# B&R Automation Studio project X20AP3x
Automation Studio 4.3.6.57 SP

## Configuration Config1

CPU , AutomationRuntime E3.10, Build 4.1.2, Vc V3.96.2

### Task classes (Cpu.sw)
```
Cyclic#1 (cycle 2000 us, tolerance 0 us):
  CondMon <- ConditionalMonitoring.CondMon.prg
Binaries: ashwd, sysconf, asfw, arconfig, iomap
Libraries: AsFltGen, AsBrStr, runtime, X20AP31x, astime, asieccon
```

### Hardware
```
PLC1 : X20CP1484 v1.1.5.0
  Connector IF2:
    ActivateDevice = 1
    Mode = Manual
    InternetAddress = 10.49.40.222
    SubnetMask = 255.255.255.0
  Connector IF3:
    InaNodeNumber = 1
  Cyclic1Duration = 2000
  Cyclic1Tolerance = 0
  Cyclic2Duration = 10000
  Cyclic2Tolerance = 10000
X20AP3131 : X20AP3131 v1.1.1.0  [SS1 -> X20TB32.SS; SL -> X20BM32.SL1]
  Supervision = off
  EnergyUnit = 1Ws
  ConfigPhaseN = calc
  VoltageWarnLim = 22000
  ZeroCrossing = on
  DisPFmeanT = off
  DisPmeanT = off
  DisQmeanT = off
  DisSmeanT = off
  DisAcEnT = off
  DisReacEnT = off
  DisAppEnT = off
  FlatStreamActivate = on
X20BM32 : X20BM32 v1.0.0.1  [X2X1 -> PLC1.IF6]
X20TB32 : X20TB32 v1.0.0.1
```

### IoMap.iom - PLC1/IoMap.iom
```iecst
(********************************************************************
 * COPYRIGHT -- Bernecker + Rainer
 ********************************************************************
 * Datei: IoMap.iom
 * Autor: hilchenbachc
 * Erstellt: 10. Januar 2014
 ********************************************************************
 * IO-Rangierungsdatei
 ********************************************************************)
VAR_CONFIG
	::CondMon:iomapping.in.InputSequence AT %IB."X20AP3131".InputSequence;
	::CondMon:iomapping.in.RxByte1 AT %IB."X20AP3131".RxByte1;
	::CondMon:iomapping.in.RxByte2 AT %IB."X20AP3131".RxByte2;
	::CondMon:iomapping.in.RxByte3 AT %IB."X20AP3131".RxByte3;
	::CondMon:iomapping.in.RxByte4 AT %IB."X20AP3131".RxByte4;
	::CondMon:iomapping.in.RxByte5 AT %IB."X20AP3131".RxByte5;
	::CondMon:iomapping.in.RxByte6 AT %IB."X20AP3131".RxByte6;
	::CondMon:iomapping.in.RxByte7 AT %IB."X20AP3131".RxByte7;
	::CondMon:iomapping.out.OutputSequence AT %QB."X20AP3131".OutputSequence;
	::CondMon:iomapping.out.EnabEnergy AT %QX."X20AP3131".EnabEnergy;
	::CondMon:iomapping.in.RBTrigDFT AT %IX."X20AP3131".RBTrigDFT;
	::CondMon:iomapping.out.TrigDFT AT %QX."X20AP3131".TrigDFT;
	::condMonData.MainsStatus.WarningPhaseA AT %IX."X20AP3131".WarningPhaseA;
	::condMonData.MainsStatus.WarningPhaseB AT %IX."X20AP3131".WarningPhaseB;
	::condMonData.MainsStatus.WarningPhaseC AT %IX."X20AP3131".WarningPhaseC;
	::condMonData.MainsStatus.LossPhaseA AT %IX."X20AP3131".LossPhaseA;
	::condMonData.MainsStatus.LossPhaseB AT %IX."X20AP3131".LossPhaseB;
	::condMonData.MainsStatus.LossPhaseC AT %IX."X20AP3131".LossPhaseC;
END_VAR
```

## Logical view

Binary libraries used (declarations not repeated): operator, runtime, astime, AsIecCon, AsBrStr, AsFltGen


### Package Logical/ConditionalMonitoring - Energieerfassung

### ConditionalMonitoring.typ - Paket Datentypen
```iecst
TYPE
	CondMonEnergy : 	STRUCT
		SVenergyT : LREAL; (* (Vector Sum) Total Apparent Energy [kWh]*)
	END_STRUCT;
	CondMonPower : 	STRUCT
		SVmeanT : LREAL; (*  (Vector Sum) Total Apparent Power [W]*)
		PmeanT : LREAL; (* Total Active Power [W]*)
		QmeanT : LREAL; (*  Total Reactive Power [W]*)
		PFmeanT : LREAL; (*  Total power factor [1]*)
	END_STRUCT;
	CondMonMainsStatus : 	STRUCT
		frequency : LREAL; (*Netzfrequenz*)
		TresholdWarning : LREAL; (*Spannungsschwelle für Warnung*)
		WarningPhaseA : BOOL;
		WarningPhaseB : BOOL;
		WarningPhaseC : BOOL;
		TresholdLoss : LREAL; (*Spannungsschwelle für Ausfall*)
		LossPhaseA : BOOL;
		LossPhaseB : BOOL;
		LossPhaseC : BOOL;
		MainsOK : BOOL;
	END_STRUCT;
	CondMonRMS : 	STRUCT
		UrmsA : LREAL; (* phase A voltage RMS [V]*)
		UrmsB : LREAL; (* phase B voltage RMS [V]*)
		UrmsC : LREAL; (* phase C voltage RMS [V]*)
		IrmsN : LREAL; (* N Line calculated current RMS [A]*)
		IrmsA : LREAL; (* phase A voltage RMS [A]*)
		IrmsB : LREAL; (* phase B voltage RMS [A]*)
		IrmsC : LREAL; (* phase C voltage RMS [A]*)
	END_STRUCT;
	CondMonData : 	STRUCT
		Rms : CondMonRMS; (*elektrische Effektivwerte*)
		Power : CondMonPower; (*elektrische Leistung*)
		Energy : CondMonEnergy; (*elektrische Arbeit*)
		MainsStatus : CondMonMainsStatus; (*Status des Versorgungsnetzes*)
	END_STRUCT;
END_TYPE
```

### ConditionalMonitoring.var - Paket Variablen
```iecst
VAR
	condMonData : CondMonData; (*Condition Monitoring*)
END_VAR
```

### Library Logical/ConditionalMonitoring/X20AP31x (ANSIC) - X20AP31x - Module- Handling via FlatStream
Depends on: AsFltGen, AsBrStr

#### X20AP31x.typ - Exportierte Datentypen
```iecst
(********************************************************************
 * COPYRIGHT -- Bernecker + Rainer
 ********************************************************************
 * Library: X20AP31x
 * Datei: X20AP31x.typ
 * Autor: B&R
 * Erstellt: 10. Januar 2014
 ********************************************************************
 * Datentypen der Library X20AP31x
 ********************************************************************)

TYPE
	X20AP31X_OUTPUT_MAPPING : 	STRUCT
		OutputSequence : USINT;
		TrigDFT : BOOL;
		EnabEnergy : BOOL;
	END_STRUCT;
	X20AP31X_INPUT_MAPPING : 	STRUCT
		InputSequence : USINT;
		RxByte1 : USINT;
		RxByte2 : USINT;
		RxByte3 : USINT;
		RxByte4 : USINT;
		RxByte5 : USINT;
		RxByte6 : USINT;
		RxByte7 : USINT;
		RBTrigDFT : BOOL;
	END_STRUCT;
	X20AP31X_MAPPING : 	STRUCT
		out : X20AP31X_OUTPUT_MAPPING;
		in : X20AP31X_INPUT_MAPPING;
	END_STRUCT;
	X20AP31X_ADC_REG_STATUS : 	STRUCT
		SysStatus0 : UINT; (*System Status 0*)
		SysStatus1 : UINT; (*System Status 1*)
		EnStatus0 : UINT; (*Metering Status 0*)
		EnStatus1 : UINT; (*Metering Status 1*)
	END_STRUCT;
	X20AP31X_ADC_REG_RMS : 	STRUCT
		IrmsN1 : UINT; (* N Line Sampled current RMS *)
		UrmsA : UINT; (* phase A voltage RMS *)
		UrmsB : UINT; (* phase B voltage RMS *)
		UrmsC : UINT; (* phase C voltage RMS *)
		IrmsN0 : UINT; (* N Line calculated current RMS *)
		IrmsA : UINT; (* phase A current RMS *)
		IrmsB : UINT; (* phase B current RMS *)
		IrmsC : UINT; (* phase C current RMS *)
	END_STRUCT;
	X20AP31X_ADC_REG_THD_ANGLE : 	STRUCT  (* THD+N, Frequency, Angle and Temperature Registers *)
		THDNUA : UINT; (* phase A voltage THD+N *)
		THDNUB : UINT; (*  phase B voltage THD+N *)
		THDNUC : UINT; (* phase C voltage THD+N *)
		THDNIA : UINT; (* phase A current THD+N *)
		THDNIB : UINT; (* phase B current THD+N *)
		THDNIC : UINT; (* phase C current THD+N *)
		Freq : UINT; (* Frequency *)
		PAngleA : INT; (* phase A mean phase angle *)
		PAngleB : INT; (* phase B mean phase angle *)
		PAngleC : INT; (* phase C mean phase angle *)
		Temp : INT; (* Measured temperature *)
		UangleA : INT; (* phase A voltage phase angle *)
		UangleB : INT; (* phase B voltage phase angle *)
		UangleC : INT; (* phase C voltage phase angle *)
	END_STRUCT;
	X20AP31X_ADC_REG_POWER : 	STRUCT  (* Power and Power Factor/ Fundamental/ Harmonic Power and Voltage/ Current RMS Registers
SVmeanTLSB: UINT;	(* LSB of (Vector Sum) Total Apparent Power *)
		SVmeanTLSB : UINT; (*LSB of (Vector Sum) Total Apparent Power

*)
		SVmeanT : UINT; (*  (Vector Sum) Total Apparent Power *)
		PmeanT : INT; (* Total Active Power *)
		PmeanA : INT; (* Phase A Active Power *)
		PmeanB : INT; (* Phase B Active Power *)
		PmeanC : INT; (* Phase C Active Power *)
		QmeanT : INT; (*  Total Reactive Power *)
		QmeanA : INT; (*  Phase A Reactive Power *)
		QmeanB : INT; (*  Phase B Reactive Power *)
		QmeanC : INT; (*  Phase C Reactive Power *)
		SAmeanT : INT; (*  (Arithmetic Sum) Total apparent power *)
		SmeanA : INT; (*  phase A apparent power *)
		SmeanB : INT; (*  phase B apparent power *)
		SmeanC : INT; (*  phase C apparent power *)
		PFmeanT : INT; (*  Total power factor *)
		PFmeanA : INT; (*  phase A power factor *)
		PFmeanB : INT; (*  phase A power factor *)
		PFmeanC : INT; (*  phase A power factor *)
		PmeanTF : INT; (*  Total active fundamental power *)
		PmeanAF : INT; (*  phase A active fundamental power *)
		PmeanBF : INT; (*  phase B active fundamental power *)
		PmeanCF : INT; (*  phase C active fundamental power *)
		PmeanTH : INT; (*  Total active harmonic power *)
		PmeanAH : INT; (* phase A active harmonic power *)
		PmeanBH : INT; (*  phase B active harmonic power *)
		PmeanCH : INT; (*  phase C active harmonic power *)
	END_STRUCT;
	X20AP31X_ADC_REG_ENERGY : 	STRUCT
		APenergyT : UDINT; (* Total Forward Active Energy *)
		APenergyA : UDINT; (*Phase A Forward Active Energy *)
		APenergyB : UDINT; (*Phase B Forward Active Energy *)
		APenergyC : UDINT; (*Phase C Forward Active Energy *)
		ANenergyT : UDINT; (*Total Reverse Active Energy *)
		ANenergyA : UDINT; (*Phase A Reverse Active Energy *)
		ANenergyB : UDINT; (*Phase B Reverse Active Energy *)
		ANenergyC : UDINT; (*Phase C Reverse Active Energy *)
		RPenergyT : UDINT; (*Total Forward Reactive Energy *)
		RPenergyA : UDINT; (*Phase A Forward Reactive Energy *)
		RPenergyB : UDINT; (*Phase B Forward Reactive Energy *)
		RPenergyC : UDINT; (*Phase C Forward Reactive Energy *)
		RNenergyT : UDINT; (*Total Reverse Reactive Energy *)
		RNenergyA : UDINT; (*Phase A Reverse Reactive Energy *)
		RNenergyB : UDINT; (*Phase B Reverse Reactive Energy *)
		RNenergyC : UDINT; (*Phase C Reverse Reactive Energy *)
		SAenergyT : UDINT; (* (Arithmetic Sum) Total Apparent Energy *)
		SenergyA : UDINT; (* Phase A Apparent Energy *)
		SenergyB : UDINT; (* Phase B Apparent Energy *)
		SenergyC : UDINT; (* Phase C Apparent Energy *)
		SVenergyT : UDINT; (* (Vector Sum) Total Apparent Energy *)
		APenergyTF : UDINT; (* Total Forward Active Fundamental Energy *)
		APenergyAF : UDINT; (* Phase A Forward Active Fundamental Energy *)
		APenergyBF : UDINT; (* Phase B Forward Active Fundamental Energy *)
		APenergyCF : UDINT; (* Phase C Forward Active Fundamental Energy *)
		ANenergyTF : UDINT; (* Total Reverse Active Fundamental Energy *)
		ANenergyAF : UDINT; (* Phase A Reverse Active Fundamental Energy *)
		ANenergyBF : UDINT; (* Phase B Reverse Active Fundamental Energy *)
		ANenergyCF : UDINT; (* Phase C Reverse Active Fundamental Energy *)
		APenergyTH : UDINT; (* Total Forward Active Harmonic Energy *)
		APenergyAH : UDINT; (* Phase A Forward Active Harmonic Energy *)
		APenergyBH : UDINT; (* Phase B Forward Active Harmonic Energy *)
		APenergyCH : UDINT; (* Phase C Forward Active Harmonic Energy *)
		ANenergyTH : UDINT; (* Total Reverse Active Harmonic Energy *)
		ANenergyAH : UDINT; (* Phase A Reverse Active Harmonic Energy *)
		ANenergyBH : UDINT; (* Phase B Reverse Active Harmonic Energy *)
		ANenergyCH : UDINT; (* Phase C Reverse Active Harmonic Energy *)
		AEnergyT : DINT; (* Total Active Energy *)
		REnergyT : DINT; (* Total Reactive Energy *)
	END_STRUCT;
	X20AP31X_ADC_REG_DFT : 	STRUCT  (*  (* Arithmetic ratio, 2 bits integer and 14 bits fractional;	That is:	Harmonic Ratio (%) = Register Value / 163.84 *)
		DftAI : ARRAY[0..31]OF UINT; (* phase A, Current, Harmonic Ratio for 2-th TO 32-th order component and Total Harmonic Distortion	Ratio *)
		DftBI : ARRAY[0..31]OF UINT; (*  phase B, Current, Harmonic Ratio for 2-th to 32-th order component and Total Harmonic Distortion	Ratio *)
		DftCI : ARRAY[0..31]OF UINT; (*  phase C, Current, Harmonic Ratio for 2-th to 32-th order component and Total Harmonic Distortion	Ratio *)
		DftAV : ARRAY[0..31]OF UINT; (*  phase A, Voltage, Harmonic Ratio for 2-th to 32-th order component and Total Harmonic Distortion	Ratio *)
		DftBV : ARRAY[0..31]OF UINT; (*  phase B, Voltage, Harmonic Ratio for 2-th to 32-th order component and Total Harmonic Distortion	Ratio *)
		DftCV : ARRAY[0..31]OF UINT; (*  phase C, Voltage, Harmonic Ratio for 2-th to 32-th order component and Total Harmonic Distortion	Ratio *) (*
		Format: Need special scaling/conversion.	The register value * 147.62 = full-scale input signal RMS.
		Current, Fundamental component value = Register Value * 209 * 65.535 / 8388608
		Voltage, Fundamental component value = Register Value * 209 * 655.35 / 8388608

	*)
		DftAI_Fund : UINT;
		DftAV_Fund : UINT;
		DftBI_Fund : UINT;
		DftBV_Fund : UINT;
		DftCI_Fund : UINT;
		DftCV_Fund : UINT;
	END_STRUCT;
	X20AP31X_ADC_REG_CFGACT : 	STRUCT  (*  Excerpt of configuration registers used by APROL, readable only by FS-IF
and with register numbers of registers with the same names. *)
		ChanControl : UINT;
		IDispTh : UINT;
		I_RatioA : UINT;
		I_RatioB : UINT;
		I_RatioC : UINT;
		I_RatioN : UINT;
		ZXConfig : UINT; (*1090*)
		SagTh : UINT; (*1094*)
		PhaseLoseTh : UINT; (*1098*)
		INWarnTh0 : UINT; (*1102*)
		INWarnTh1 : UINT; (*1106*)
		THDNUTh : UINT; (*1110*)
		THDNITh : UINT; (*1114*)
		MeteringMode : UINT; (*MeteringMode 1162*)
		PLconst : UDINT; (*Powerline Constant*)
	END_STRUCT;
	X20AP31X_ENV_STATUS : 	STRUCT  (* Environment Variables *)
		ulUpTime : UDINT;
		ulUpCnt : UDINT;
		ssMinTemp : INT;
		ssMaxTemp : INT;
		ulRes : ARRAY[0..12]OF UDINT;
	END_STRUCT;
	X20AP31X : 	STRUCT
		NetTimeReg : UDINT; (* TIME OF Section copy TO Buffer *)
		Status : X20AP31X_ADC_REG_STATUS; (* Status registers *)
		Rms : X20AP31X_ADC_REG_RMS; (* RMS Registers *)
		Power : X20AP31X_ADC_REG_POWER; (* Power Registers *)
		ThdAngle : X20AP31X_ADC_REG_THD_ANGLE; (* THD + Angel Registers *)
		NetTimeEnergy : UDINT; (* TIME OF Section copy TO Buffer *)
		Energy : X20AP31X_ADC_REG_ENERGY; (* Energy Registers *)
		NetTimeDft : UDINT; (* TIME OF Section copy TO Buffer *)
		Dft : X20AP31X_ADC_REG_DFT; (* DFT Registers *)
		CfgAct : X20AP31X_ADC_REG_CFGACT; (* Config read back *)
		EnvReg : X20AP31X_ENV_STATUS; (* Read Back Environment Registers *)
	END_STRUCT;
END_TYPE
```

#### X20AP31x.fun - Exportierte Funktionen und Funktionsblöcke
```iecst
FUNCTION_BLOCK X20AP31X_Register (*Read X20AP3X1 - Register*)
	VAR_INPUT
		pMapping : REFERENCE TO X20AP31X_MAPPING; (*Pointer to IO-Mapping- Datetype*)
		pData : REFERENCE TO X20AP31X; (*Pointer to Module Data*)
	END_VAR
	VAR
		read : fltRead;
		write : fltWrite;
		fltMTUWrite : ARRAY[0..3] OF USINT;
		fltMTURead : ARRAY[0..7] OF USINT;
		blockNumber : USINT;
		blockReceived : USINT;
		tmpBuf : ARRAY[0..799] OF SINT;
	END_VAR
END_FUNCTION_BLOCK
```

#### X20AP31X_Register.c - Read X20AP3X1 - Register
```c
/********************************************************************
 * COPYRIGHT -- Bernecker + Rainer
 ********************************************************************
 * Library: X20AP31x
 * Datei: X20AP31X_Register.c
 * Autor: B&R
 * Erstellt: 10. Januar 2014
 ********************************************************************
 * Implementierung der Library X20AP31x
 ********************************************************************/

#include <bur/plctypes.h>
#ifdef __cplusplus
	extern "C"
	{
#endif

	#include "X20AP31x.h"

#ifdef __cplusplus
	};
#endif

/* Read X20AP3X1 - Register */
void X20AP31X_Register(struct X20AP31X_Register* inst)
{

		inst->pMapping->out.EnabEnergy = 1;

		// cyclically trigger generation of Energy and DFT values on AP31x1
		if (  inst->pMapping->in.RBTrigDFT == inst->pMapping->out.TrigDFT )
		{
			inst->pMapping->out.TrigDFT ^= 1;
		}

		// copy Inputs to Read Buffer //
		inst->fltMTURead[0] = inst->pMapping->in.InputSequence;
		inst->fltMTURead[1] = inst->pMapping->in.RxByte1;
		inst->fltMTURead[2] = inst->pMapping->in.RxByte2;
		inst->fltMTURead[3] = inst->pMapping->in.RxByte3;
		inst->fltMTURead[4] = inst->pMapping->in.RxByte4;
		inst->fltMTURead[5] = inst->pMapping->in.RxByte5;
		inst->fltMTURead[6] = inst->pMapping->in.RxByte6;
		inst->fltMTURead[7] = inst->pMapping->in.RxByte7;

		// Flat Stream Handling

		inst->read.enable	 		= 1;
		inst->read.cfg		 	= fltMODE_FRAME;
		inst->read.pBuf			= (UDINT)&inst->tmpBuf;
		inst->read.bufLen			= sizeof(inst->tmpBuf);
		inst->read.pRxBytes	 	= (UDINT)&inst->fltMTURead[0];
		inst->read.rxBytesLen 	= sizeof(inst->fltMTURead);
		fltRead(&inst->read);
		if (inst->read.status == fltERR_FRAME_FINISHED)
		{
			int len;

			if ((len = inst->read.validBytes) != 0)
			{

				inst->blockReceived = inst->tmpBuf[0];
				len	= sizeof(X20AP31X);

				if (len > inst->read.validBytes)
					len = inst->read.validBytes;

				brsmemcpy ( (UDINT) inst->pData, (UDINT) &inst->tmpBuf[1], len);
			}
		}

		inst->write.enable	 	= 1;
		inst->write.cfg			= 	(fltMODE_SYNCHRON + (1 << 4) + (1 << 1));
		inst->write.readSequ 		= inst->read.readSequ;
		inst->write.pBuf			= (UDINT)&inst->blockNumber;
		inst->write.bufLen		= 0;
		inst->write.pTxBytes		= (UDINT)&inst->fltMTUWrite[0];
		inst->write.txBytesLen	= sizeof(inst->fltMTUWrite);
		inst->write.pSequ	 		= (UDINT)&inst->fltMTURead[0];
		fltWrite(&inst->write);
		if (inst->write.status == 0)
		{

		}

		/* copy write buffer to outputs */
		inst->pMapping->out.OutputSequence = inst->fltMTUWrite[0];

}
```

### Program Logical/ConditionalMonitoring/CondMon (IEC) - Ein neues Programm

#### CondMon.st - Implementierungscode
```iecst
(********************************************************************
 * COPYRIGHT -- Bernecker + Rainer
 ********************************************************************
 * Programm: energy
 * Datei: energy.st
 * Autor: B&R
 * Erstellt: 16. Januar 2014
 ********************************************************************
 * Implementierung des Programms energy
 ********************************************************************)

PROGRAM _INIT

fubAP31x.pData := ADR(apData);
fubAP31x.pMapping := ADR(iomapping);
converterRatio := 50/5; 	(* tatsächlich verwendeter Stromwandler *)

END_PROGRAM

PROGRAM _CYCLIC

(*  ----------------------------------------------------------------------------------------
	Korrekturfaktor, da nicht alle Stromwandler- Übersetzungen im Modul konfigurierbar sind.
	Es wird dabei davon ausgegangen, dass alle Phasen den gleichen Übersetzungsfaktor haben.
	----------------------------------------------------------------------------------------
*)
currentCorrectionFactor := converterRatio / (UINT_TO_LREAL(apData.CfgAct.I_RatioA) / 10);

(* Daten aus dem X20AP- Modul abrufen *)
fubAP31x();

(*  ----------------------------------------------------------------------------------------
	Effektivwerte der Ströme und Spannungen.
	----------------------------------------------------------------------------------------
*)
(* Stromwerte werden vom Modul in 0,001 A geliefert *)
condMonData.Rms.IrmsA := UINT_TO_LREAL(apData.Rms.IrmsA) * currentCorrectionFactor / 1000.0;
condMonData.Rms.IrmsB := UINT_TO_LREAL(apData.Rms.IrmsB) * currentCorrectionFactor / 1000.0;
condMonData.Rms.IrmsC := UINT_TO_LREAL(apData.Rms.IrmsC) * currentCorrectionFactor / 1000.0;
condMonData.Rms.IrmsN := UINT_TO_LREAL(apData.Rms.IrmsN0) * currentCorrectionFactor / 1000.0;
(* Spannungswerte werden vom Modul in 0,01 V geliefert *)
condMonData.Rms.UrmsA := UINT_TO_LREAL(apData.Rms.UrmsA) / 100.0;
condMonData.Rms.UrmsB := UINT_TO_LREAL(apData.Rms.UrmsB) / 100.0;
condMonData.Rms.UrmsC := UINT_TO_LREAL(apData.Rms.UrmsC) / 100.0;

(*  ----------------------------------------------------------------------------------------
	Leistung
	----------------------------------------------------------------------------------------
*)
(* Gesamt- Leistungswerte werden vom Modul in 4W- Schritten geliefert *)
condMonData.Power.SVmeanT := ( UINT_TO_LREAL(apData.Power.SVmeanT) + UINT_TO_LREAL(apData.Power.SVmeanTLSB)/65536 ) * 4.0 * currentCorrectionFactor;
condMonData.Power.PmeanT := INT_TO_LREAL(apData.Power.PmeanT) * 4.0 * currentCorrectionFactor;
condMonData.Power.QmeanT := INT_TO_LREAL(apData.Power.QmeanT) * 4.0 * currentCorrectionFactor;
(* Leistungsfaktor wird vom Modul in 0,001 - Einheiten geliefert *)
condMonData.Power.PFmeanT := INT_TO_LREAL(apData.Power.PFmeanT) / 1000.0;

(*  ----------------------------------------------------------------------------------------
	Arbeit
	----------------------------------------------------------------------------------------
*)
(* Energie wird in 0,1 oder 0,01 CF geliefert *)
IF apData.CfgAct.PLconst <> 0 THEN
	unitsPerkWh := 3600.0 * (1250000000.0 / apData.CfgAct.PLconst);
	IF apData.CfgAct.MeteringMode.3 THEN
		unitsPerkWh := unitsPerkWh * 10.0;
	END_IF
ELSE
	unitsPerkWh := 0;
END_IF
condMonData.Energy.SVenergyT := UDINT_TO_LREAL(apData.Energy.SVenergyT) / unitsPerkWh * currentCorrectionFactor;

(*  ----------------------------------------------------------------------------------------
	Netzüberwachung
	----------------------------------------------------------------------------------------
*)

condMonData.MainsStatus.TresholdWarning := UINT_TO_LREAL(apData.CfgAct.SagTh) / 100.0;
condMonData.MainsStatus.TresholdLoss := UINT_TO_LREAL(apData.CfgAct.PhaseLoseTh) / 100.0;
condMonData.MainsStatus.frequency := UINT_TO_LREAL(apData.ThdAngle.Freq) / 100.0;
condMonData.MainsStatus.MainsOK := NOT(condMonData.MainsStatus.LossPhaseA) AND NOT(condMonData.MainsStatus.LossPhaseB) AND NOT(condMonData.MainsStatus.LossPhaseC) AND
								   NOT(condMonData.MainsStatus.WarningPhaseA) AND NOT(condMonData.MainsStatus.WarningPhaseB) AND NOT(condMonData.MainsStatus.WarningPhaseC);

END_PROGRAM
```

#### CondMon.var - Lokale Variablen
```iecst
(********************************************************************
 * COPYRIGHT -- Bernecker + Rainer
 ********************************************************************
 * Programm: energy
 * Datei: energy.var
 * Autor: hilchenbachc
 * Erstellt: 16. Januar 2014
 ********************************************************************
 * Lokale Variablen des Programms energy
 ********************************************************************)
VAR
	iomapping : X20AP31X_MAPPING; (*IO- Mapping für X20AP3x - Module*)
	apData : X20AP31X; (*Ausgabedaten für X20AP3x- Module*)
	fubAP31x : X20AP31X_Register; (*Funktionsbaustein zum Lesen der X20AP3X- Module*)
	converterRatio : LREAL; (*Übersetzungsverhältnis des Stromwandlers*)
	currentCorrectionFactor : LREAL;
	unitsPerkWh : LREAL;
END_VAR
```

### X20AP3131_IO_Konfiguration.txt
```
IF6.ST1			X20AP3131
 Funktionsmodell	Standard		Arbeitsweise des Moduls
 Allgemein
  Modulueberwachung	Aus		Service Mode ausloesen, wenn Modul nicht vorhanden ist
 Allgemeine Einstellungen
  Netzanschaltung	Einzel- / Drei-Phasen Messung		Auswahl Anschaltung durch Anzahl der gemessenen Phasen
  Netzwerkfrequenz	50		Auswahl Frequenz [Hz]
  Energie-Einheit	[1Ws]		Auswahl Energie-Einheit
  Stromschwelle LED ein	100		Legt die Stromschwelle fest [mA]
  Format der Status- und Controlinformation	Einzelvariablen		Auswahl Darstellungsart
 Physikalische Netzwerkeinstellungen
  Phase A	Ein
  Phase A Stromuebersetzungsverhaeltnis	100		Legt das Stromuebersetzungsverhaeltnis fest [0,1]
  Phase B	Ein
  Phase B Stromuebersetzungsverhaeltnis	100		Legt das Stromuebersetzungsverhaeltnis fest [0,1]
  Phase C	Ein
  Phase C Stromuebersetzungsverhaeltnis	100		Legt das Stromuebersetzungsverhaeltnis fest [0,1]
  Nullleiter N	Berechnung		Auswahl gemessener oder berechneter Strom
  Nullleiter N Stromueberwachung	Aus		De-/aktiviere Statusueberwachung und Anzeige
  Nullleiter N Strom-Alarmschwelle	50		Legt die Alarmschwelle fest [mA]
 Einstellungen Warnung- und Ausfallschwellwerte
  Spannungsschwellwerte	Ein		De-/Aktiviere Konfiguration und Statusinformation
  Schwelle Spannungswarnung	22000		Effektivwert [0,01 V]
  Schwelle Spannungsausfall	2500		Effektivwert [0,01 V]
  Schwelle Oberwellenspannungswarnung	1000		Wert [0,01 %]
  Schwelle Oberwellenstromwarnung	1000		Wert [0,01 %]
  Format der Statusinformation	Einzelvariablen		Auswahl Darstellungsart
 Einstellungen Nulldurchgangssignale
  Nulldurchgangssignale	Aus		De-/Aktiviere Signale
 Anzeigekonfiguration Analogwerte
  Applikationsauswahl	Einfache Leistungs-/Energiedaten
  Spannung Phase A RMS	Aus
  Spannung Phase B RMS	Aus
  Spannung Phase C RMS	Aus
  Strom Phase A RMS	Aus
  Strom Phase B RMS	Aus
  Strom Phase C RMS	Aus
  Strom Nullleiter N RMS	Aus
  Frequenz gemessen	Aus
  Leistungsfaktor gesamt	Aus
  Wirkleistung gesamt	Aus
  Blindleistung gesamt	Aus
  Scheinleistung gesamt	Aus
  Wirkenergie gesamt	Aus
  Blindenergie gesamt	Aus
  Scheinenergie gesamt - arithmetische Summe	Aus
  Scheinenergie gesamt - komplexe Summe	Aus
  System Status Selektion	Einzelvariablen
 Flat Stream Konfiguration
  User Interface Flat Stream akitivieren	Ein
  OutputMTU	off		Sendeblockgroeße [Byte]
  InputMTU	7 Byte		Empfangsblockgroeße [Byte]
  BlockForward	1		Anzahl der abgesendeten Bloecke ohne Bestaetigung
  BlockForward Verzoegerungszeit	0		Zusaetzliche Verzoegerungszeit zwischen zwei unbestaetigt gesendeten Bloecken[usec]
  Mehrfachsegmente	Aus		Mehrfachsegmente innerhalb MTU moeglich
  Segmentgroeße	Aus		Segmentgroeße darf MTU ueberschreiten
 Simulation
  Simulationsgeraet			Zugeordnetes Simulationsgeraet
```

Listed in the project but not available here: Logical/ConditionalMonitoring/X20AP31x/X20AP31x.var
